// TIA Portal V20 export
FUNCTION_BLOCK "FB_DataLog"   // FB10, LAD
{ S7_Optimized_Access := 'TRUE' }
// stored: AutoNumber false, MemoryReserve 100, SetENOAutomatically false
   VAR_INPUT
      DataLogCreate_REQ : Bool;
      DataLogOpen_REQ : Bool;
      DataLogWrite_REQ : Bool;
      DataLogClose_REQ : Bool;
      DataLogClear_REQ : Bool;
      DataLogDelete_REQ : Bool;
   END_VAR
   VAR_OUTPUT
      DataLogCreate_DONE : Bool;
      DataLogCreate_BUSY : Bool;
      DataLogCreate_ERROR : Bool;
      DataLogCreate_STATUS : Word;
      DataLogOpen_DONE : Bool;
      DataLogOpen_BUSY : Bool;
      DataLogOpen_ERROR : Bool;
      DataLogOpen_STATUS : Word;
      DataLogWrite_DONE : Bool;
      DataLogWrite_BUSY : Bool;
      DataLogWrite_ERROR : Bool;
      DataLogWrite_STATUS : Word;
      DataLogClose_DONE : Bool;
      DataLogClose_BUSY : Bool;
      DataLogClose_ERROR : Bool;
      DataLogClose_STATUS : Word;
      DataLogClear_DONE : Bool;
      DataLogClear_BUSY : Bool;
      DataLogClear_ERROR : Bool;
      DataLogClear_STATUS : Word;
      DataLogDelete_DONE : Bool;
      DataLogDelete_BUSY : Bool;
      DataLogDelete_ERROR : Bool;
      DataLogDelete_STATUS : Word;
   END_VAR
   VAR_IN_OUT
      ID : DWord;
      "NAME" : Variant;
      DataLogCreate_HEADER : Variant;
      DATA : Variant;
   END_VAR
   VAR
      Enable_DataLogOpen : Bool;
      Enable_DataLogWrite : Bool;
      Axiliar_P_Trig_0 : Bool;
      Axiliar_P_Trig_1 : Bool;
      Axiliar_P_Trig_2 : Bool;
      Axiliar_P_Trig_3 : Bool;
      Axiliar_P_Trig_4 : Bool;
      Axiliar_P_Trig_5 : Bool;
      Axiliar_P_Trig_6 : Bool;
      Axiliar_P_Trig_7 : Bool;
      Axiliar_P_Trig_8 : Bool;
      DataLogCreate_Instance { S7_SetPoint := 'True'} : DataLogCreate;
      DataLogOpen_Instance { S7_SetPoint := 'True'} : DataLogOpen;
      DataLogWrite_Instance { S7_SetPoint := 'True'} : DataLogWrite;
      DataLogClose_Instance { S7_SetPoint := 'True'} : DataLogClose;
      DataLogClear_Instance { S7_SetPoint := 'True'} : DataLogClear;
      DataLogDelete_Instance { S7_SetPoint := 'True'} : DataLogDelete;
   END_VAR
   VAR_TEMP   // added for the SCL form of the ladder/FBD networks
      _w1 : Bool;
      _w2 : Bool;
      _w3 : Bool;
   END_VAR
BEGIN

REGION Network 1: Create DataLog
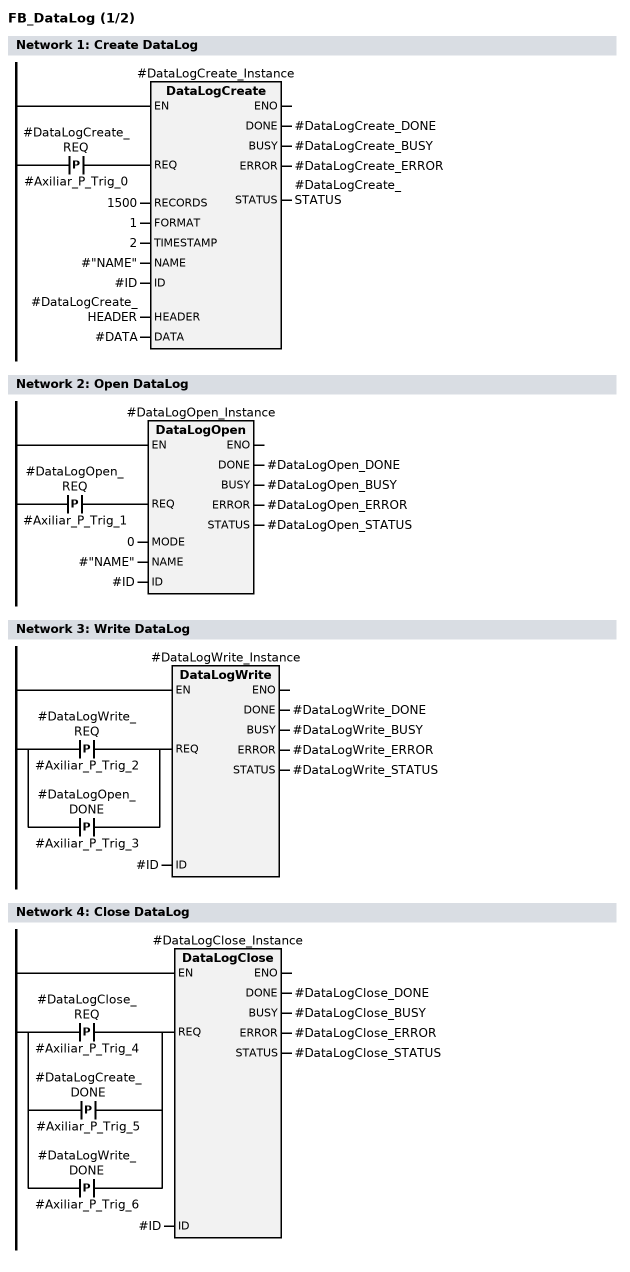
   RUNG wire#powerrail
      #DataLogCreate_Instance.DataLogCreate(REQ := wire#w1, RECORDS := 1500, FORMAT := 1, TIMESTAMP := 2, "NAME" := #"NAME", ID := #ID, HEADER := #DataLogCreate_HEADER, DATA := #DATA, DONE => #DataLogCreate_DONE, BUSY => #DataLogCreate_BUSY, ERROR => #DataLogCreate_ERROR, STATUS => #DataLogCreate_STATUS)
   END_RUNG
   RUNG wire#powerrail
      P_Contact(operand := #DataLogCreate_REQ, bit := #Axiliar_P_Trig_0)
   END_RUNG wire#w1
   // the same network as SCL:
   #_w1 := #DataLogCreate_REQ AND NOT #Axiliar_P_Trig_0;   // rising edge of #DataLogCreate_REQ
   #Axiliar_P_Trig_0 := #DataLogCreate_REQ;
   #DataLogCreate_Instance(REQ := #_w1,   // DataLogCreate
                           RECORDS := 1500,
                           FORMAT := 1,
                           TIMESTAMP := 2,
                           "NAME" := #"NAME",
                           ID := #ID,
                           HEADER := #DataLogCreate_HEADER,
                           DATA := #DATA,
                           DONE => #DataLogCreate_DONE,
                           BUSY => #DataLogCreate_BUSY,
                           ERROR => #DataLogCreate_ERROR,
                           STATUS => #DataLogCreate_STATUS);
END_REGION

REGION Network 2: Open DataLog
   RUNG wire#powerrail
      { S7_Templates := "card := 0" } #DataLogOpen_Instance.DataLogOpen(REQ := wire#w1, MODE := 0, "NAME" := #"NAME", ID := #ID, DONE => #DataLogOpen_DONE, BUSY => #DataLogOpen_BUSY, ERROR => #DataLogOpen_ERROR, STATUS => #DataLogOpen_STATUS)
   END_RUNG
   RUNG wire#powerrail
      P_Contact(operand := #DataLogOpen_REQ, bit := #Axiliar_P_Trig_1)
   END_RUNG wire#w1
   // the same network as SCL:
   #_w1 := #DataLogOpen_REQ AND NOT #Axiliar_P_Trig_1;   // rising edge of #DataLogOpen_REQ
   #Axiliar_P_Trig_1 := #DataLogOpen_REQ;
   #DataLogOpen_Instance(REQ := #_w1,   // DataLogOpen
                         MODE := 0,
                         "NAME" := #"NAME",
                         ID := #ID,
                         DONE => #DataLogOpen_DONE,
                         BUSY => #DataLogOpen_BUSY,
                         ERROR => #DataLogOpen_ERROR,
                         STATUS => #DataLogOpen_STATUS);
END_REGION

REGION Network 3: Write DataLog
   RUNG wire#powerrail
      #DataLogWrite_Instance.DataLogWrite(REQ := wire#w1, ID := #ID, DONE => #DataLogWrite_DONE, BUSY => #DataLogWrite_BUSY, ERROR => #DataLogWrite_ERROR, STATUS => #DataLogWrite_STATUS)
   END_RUNG
   RUNG wire#powerrail
      P_Contact(operand := #DataLogWrite_REQ, bit := #Axiliar_P_Trig_2)
   END_RUNG wire#w1
   RUNG wire#powerrail
      P_Contact(operand := #DataLogOpen_DONE, bit := #Axiliar_P_Trig_3)
   END_RUNG wire#w1
   // the same network as SCL:
   #_w1 := #DataLogWrite_REQ AND NOT #Axiliar_P_Trig_2;   // rising edge of #DataLogWrite_REQ
   #Axiliar_P_Trig_2 := #DataLogWrite_REQ;
   #_w2 := #DataLogOpen_DONE AND NOT #Axiliar_P_Trig_3;   // rising edge of #DataLogOpen_DONE
   #Axiliar_P_Trig_3 := #DataLogOpen_DONE;
   #DataLogWrite_Instance(REQ := #_w1 OR #_w2,   // DataLogWrite
                          ID := #ID,
                          DONE => #DataLogWrite_DONE,
                          BUSY => #DataLogWrite_BUSY,
                          ERROR => #DataLogWrite_ERROR,
                          STATUS => #DataLogWrite_STATUS);
END_REGION

REGION Network 4: Close DataLog
   RUNG wire#powerrail
      #DataLogClose_Instance.DataLogClose(REQ := wire#w1, ID := #ID, DONE => #DataLogClose_DONE, BUSY => #DataLogClose_BUSY, ERROR => #DataLogClose_ERROR, STATUS => #DataLogClose_STATUS)
   END_RUNG
   RUNG wire#powerrail
      P_Contact(operand := #DataLogClose_REQ, bit := #Axiliar_P_Trig_4)
   END_RUNG wire#w1
   RUNG wire#powerrail
      P_Contact(operand := #DataLogCreate_DONE, bit := #Axiliar_P_Trig_5)
   END_RUNG wire#w1
   RUNG wire#powerrail
      P_Contact(operand := #DataLogWrite_DONE, bit := #Axiliar_P_Trig_6)
   END_RUNG wire#w1
   // the same network as SCL:
   #_w1 := #DataLogClose_REQ AND NOT #Axiliar_P_Trig_4;   // rising edge of #DataLogClose_REQ
   #Axiliar_P_Trig_4 := #DataLogClose_REQ;
   #_w2 := #DataLogCreate_DONE AND NOT #Axiliar_P_Trig_5;   // rising edge of #DataLogCreate_DONE
   #Axiliar_P_Trig_5 := #DataLogCreate_DONE;
   #_w3 := #DataLogWrite_DONE AND NOT #Axiliar_P_Trig_6;   // rising edge of #DataLogWrite_DONE
   #Axiliar_P_Trig_6 := #DataLogWrite_DONE;
   #DataLogClose_Instance(REQ := #_w1 OR #_w2 OR #_w3,   // DataLogClose
                          ID := #ID,
                          DONE => #DataLogClose_DONE,
                          BUSY => #DataLogClose_BUSY,
                          ERROR => #DataLogClose_ERROR,
                          STATUS => #DataLogClose_STATUS);
END_REGION

REGION Network 5: Clear DataLog
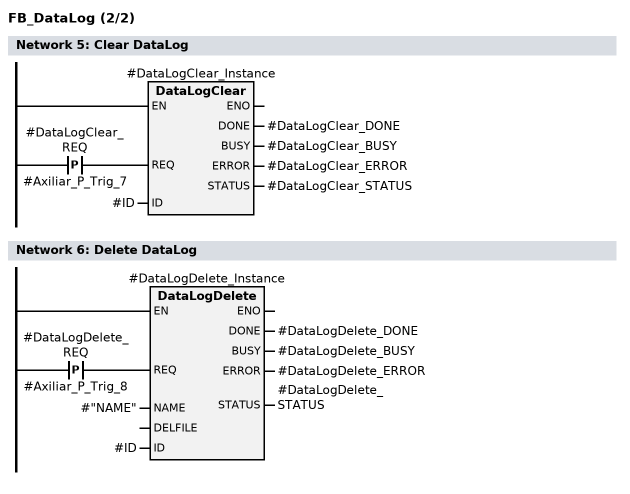
   RUNG wire#powerrail
      #DataLogClear_Instance.DataLogClear(REQ := wire#w1, ID := #ID, DONE => #DataLogClear_DONE, BUSY => #DataLogClear_BUSY, ERROR => #DataLogClear_ERROR, STATUS => #DataLogClear_STATUS)
   END_RUNG
   RUNG wire#powerrail
      P_Contact(operand := #DataLogClear_REQ, bit := #Axiliar_P_Trig_7)
   END_RUNG wire#w1
   // the same network as SCL:
   #_w1 := #DataLogClear_REQ AND NOT #Axiliar_P_Trig_7;   // rising edge of #DataLogClear_REQ
   #Axiliar_P_Trig_7 := #DataLogClear_REQ;
   #DataLogClear_Instance(REQ := #_w1,   // DataLogClear
                          ID := #ID,
                          DONE => #DataLogClear_DONE,
                          BUSY => #DataLogClear_BUSY,
                          ERROR => #DataLogClear_ERROR,
                          STATUS => #DataLogClear_STATUS);
END_REGION

REGION Network 6: Delete DataLog
   RUNG wire#powerrail
      #DataLogDelete_Instance.DataLogDelete(REQ := wire#w1, "NAME" := #"NAME", DelFile :=, ID := #ID, DONE => #DataLogDelete_DONE, BUSY => #DataLogDelete_BUSY, ERROR => #DataLogDelete_ERROR, STATUS => #DataLogDelete_STATUS)
   END_RUNG
   RUNG wire#powerrail
      P_Contact(operand := #DataLogDelete_REQ, bit := #Axiliar_P_Trig_8)
   END_RUNG wire#w1
   // the same network as SCL:
   #_w1 := #DataLogDelete_REQ AND NOT #Axiliar_P_Trig_8;   // rising edge of #DataLogDelete_REQ
   #Axiliar_P_Trig_8 := #DataLogDelete_REQ;
   #DataLogDelete_Instance(REQ := #_w1,   // DataLogDelete
                           "NAME" := #"NAME",
                           ID := #ID,
                           DONE => #DataLogDelete_DONE,
                           BUSY => #DataLogDelete_BUSY,
                           ERROR => #DataLogDelete_ERROR,
                           STATUS => #DataLogDelete_STATUS);
END_REGION
END_FUNCTION_BLOCK
